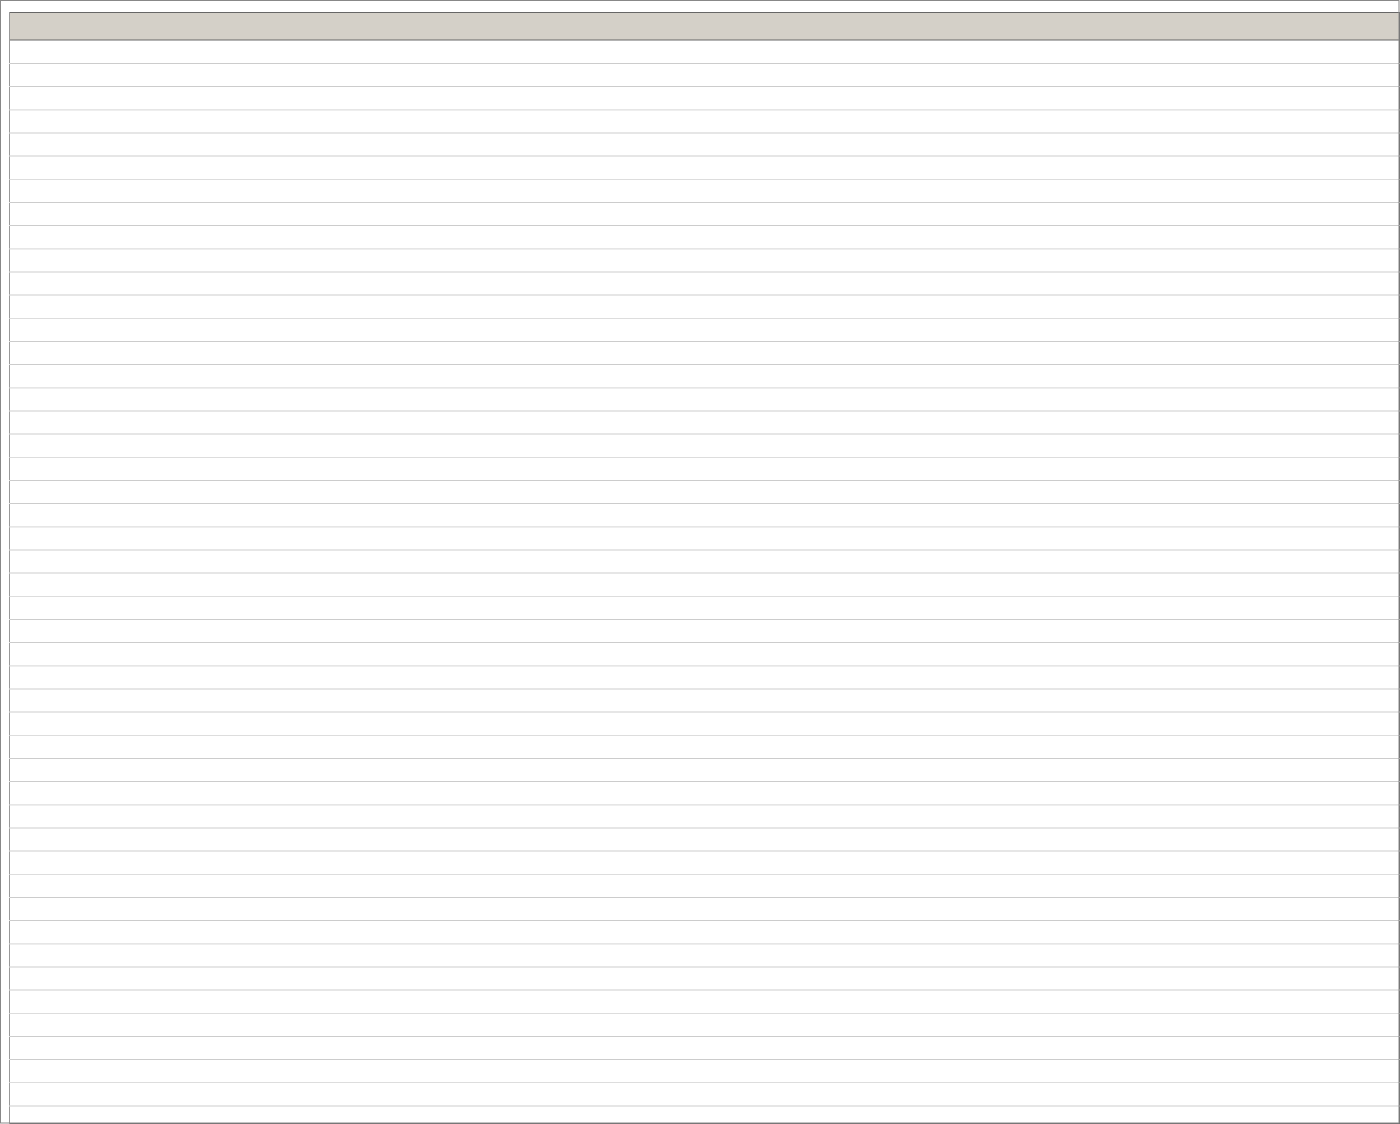
VISUALIZATION T_MESSAGE_LIST  // 1510x1213
    Table (10,13 1500x1200), data array: MessageData.VisuList
        p1128707560: GVL_AXIS_CTRL.MAX_MESSAGE
        p3854506369: MessageData.VisuList[INDEX].eType
        p1892666644: MessageData.VisuList[INDEX].eDevice
        p338671338: MessageData.VisuList[INDEX].eSubdevice
        p2170511999: MessageData.VisuList[INDEX].iErrorNumber
        p3723444502: MessageData.VisuList[INDEX].tTime
        p1218418051: MessageData.VisuList[INDEX].sText
END_VISUALIZATION

(* stored: Version 1.1.0.1, ProductVersion 3.1.4026.12
   Visu T_MESSAGE_LIST: Id {9c4a821c-b076-4bb3-9aa7-2ce8309ed9ce} *)
